PROGRAM MAIN
VAR
	BottleTester : fb_BottleTester_Main;
END_VAR

BottleTester ();

END_PROGRAM

(* stored: Version 1.1.0.1
   POU MAIN: Id {536f4be8-81f7-40ac-8d65-f08f40282c1a}, SpecialFunc None *)
